# EPICS autosave request: support/calc/2-7/calcApp/Db/interp_settings.req
$(P)interp_mode
$(P)interp.VALA
$(P)interp.VALB
$(P)interp.VALC
$(P)interp.VALN
$(P)interp_n
$(P)interp_x
$(P)interp_y1
$(P)interp_y2
